(* Logix 5000 project; controller Machine_Maintenance_Lab2 vendor 1 type 14 code 155 rev 36.11; software revision 36.00 *)

TASK MainTask (continuous, watchdog 500 ms) : MainProgram

MODULES
   Local : vendor 1 type 14 code 155 (PointIO 0, rev 36.11)
      Discrete_IO : Embedded (PointIO 1, rev 36.11, Output RPI 20 ms)
END_MODULES

PROGRAM MainProgram   (* main routine MainRoutine *)
VAR
   counter : COUNTER := (PRE := 5);
   i_CycleDone : ALIAS FOR o_CycleDone;
   i_GreenPB : ALIAS FOR Local:1:I.Data.0;
   i_GreenPB_ConveyorStart : ALIAS FOR i_GreenPB;
   i_GreenPBLight_Conveyor1ON : ALIAS FOR o_GreenPBLight_Conveyor1ON;
   i_Pause : ALIAS FOR Pause;
   i_Piston : ALIAS FOR Local:1:O.Data.2;
   i_RedPB_StopButton : ALIAS FOR Local:1:I.Data.1;
   i_RedPBLight_Conveyor2ON : ALIAS FOR o_RedPBLight_Conveyor2ON;
   i_Turnkey : ALIAS FOR Local:1:I.Data.2;
   i_Turnkey_ItemSensor : ALIAS FOR i_Turnkey;
   ItemCounter1 : COUNTER := (PRE := 5);
   ItemCounterLeft : COUNTER := (PRE := 5);
   ItemCounterRight : COUNTER := (PRE := 6);
   o_CycleDone : BOOL;
   o_GreenPBLight : ALIAS FOR Local:1:O.Data.0;
   o_GreenPBLight_Conveyor1ON : ALIAS FOR o_GreenPBLight;
   o_Piston : ALIAS FOR i_Piston;
   o_RedPBLight : ALIAS FOR Local:1:O.Data.1;
   o_RedPBLight_Conveyor2ON : ALIAS FOR o_RedPBLight;
   OS_Out : BOOL;
   Pause : BOOL;
   ResetDelay : TIMER := (PRE := 500);
   ThreeSecTimer : TIMER := (PRE := 3000);
   timer : TIMER := (PRE := 5000);
   TurnkeyOneShot : BOOL;
END_VAR

ROUTINE MainRoutine   (* ladder *)
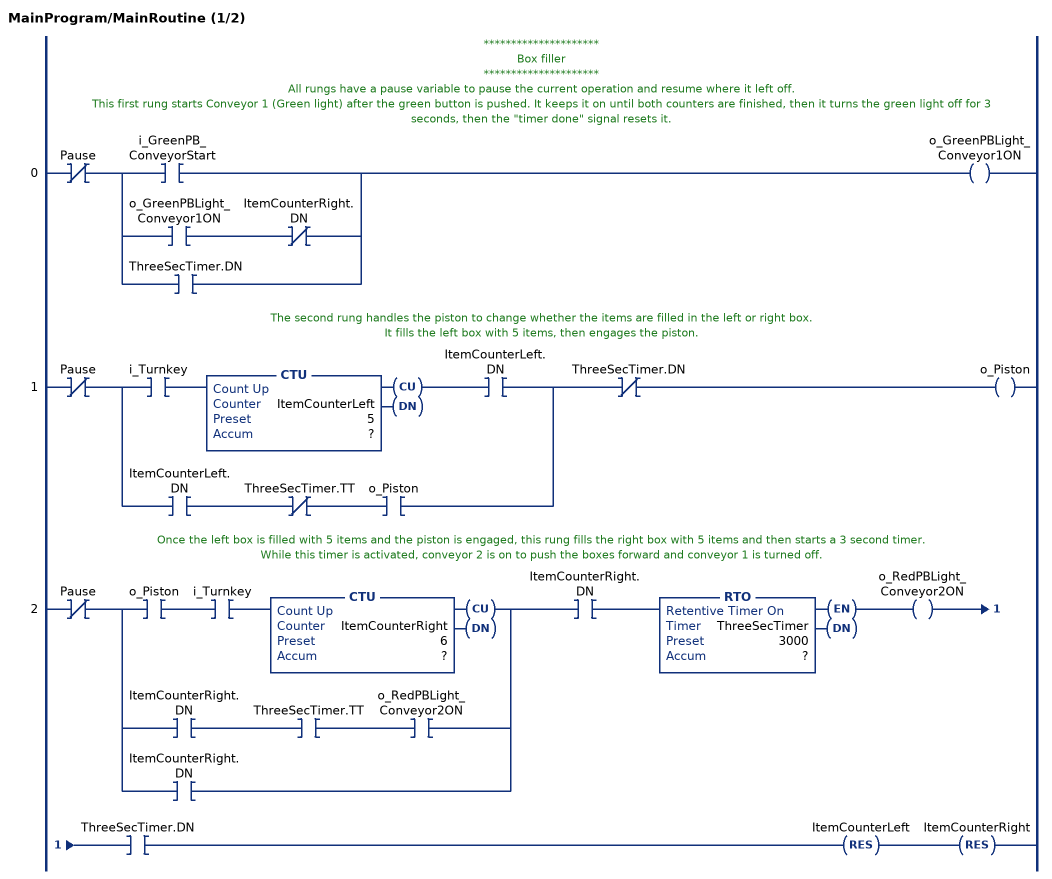
   // *********************
   // Box filler
   // *********************
   // All rungs have a pause variable to pause the current operation and resume where it left off.
   // This first rung starts Conveyor 1 (Green light) after the green button is pushed. It keeps it on until both counters are finished, then it turns the green light off for 3 seconds, then the "timer done" signal resets it.
   0: XIO(Pause)[XIC(i_GreenPB_ConveyorStart) ,[XIC(o_GreenPBLight_Conveyor1ON) XIO(ItemCounterRight.DN) ,XIC(ThreeSecTimer.DN) ] ]OTE(o_GreenPBLight_Conveyor1ON);
   // The second rung handles the piston to change whether the items are filled in the left or right box.
   // It fills the left box with 5 items, then engages the piston.
   1: XIO(Pause)[XIC(i_Turnkey) CTU(ItemCounterLeft,?,?) XIC(ItemCounterLeft.DN) ,XIC(ItemCounterLeft.DN) XIO(ThreeSecTimer.TT) XIC(o_Piston) ]XIO(ThreeSecTimer.DN)OTE(o_Piston);
   // Once the left box is filled with 5 items and the piston is engaged, this rung fills the right box with 5 items and then starts a 3 second timer.
   // While this timer is activated, conveyor 2 is on to push the boxes forward and conveyor 1 is turned off.
   2: XIO(Pause)[XIC(o_Piston) XIC(i_Turnkey) CTU(ItemCounterRight,?,?) ,[XIC(ItemCounterRight.DN) XIC(ThreeSecTimer.TT) XIC(o_RedPBLight_Conveyor2ON) ,XIC(ItemCounterRight.DN) ] ]XIC(ItemCounterRight.DN)RTO(ThreeSecTimer,?,?)OTE(o_RedPBLight_Conveyor2ON)XIC(ThreeSecTimer.DN)RES(ItemCounterLeft)RES(ItemCounterRight);
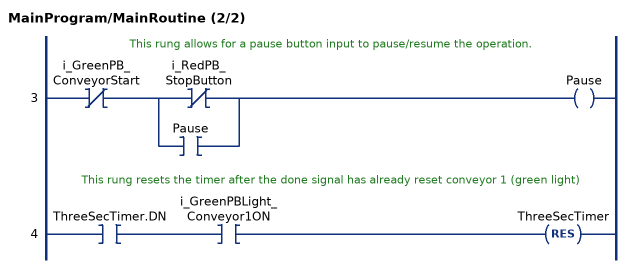
   // This rung allows for a pause button input to pause/resume the operation.
   3: XIO(i_GreenPB_ConveyorStart)[XIO(i_RedPB_StopButton) ,XIC(Pause) ]OTE(Pause);
   // This rung resets the timer after the done signal has already reset conveyor 1 (green light)
   4: XIC(ThreeSecTimer.DN)XIC(i_GreenPBLight_Conveyor1ON)RES(ThreeSecTimer);
END_ROUTINE
END_PROGRAM
